FUNCTION TryConvert_BYTE_TO_TOD : BOOL
VAR_INPUT
	in : BYTE;
	out : REFERENCE TO TOD;
END_VAR

out := BYTE_TO_TOD(in);
TryConvert_BYTE_TO_TOD := TRUE;

END_FUNCTION

(* stored: Version 1.1.0.1, ProductVersion 3.1.4024.12
   POU TryConvert_BYTE_TO_TOD: Id {392e3d4e-3f2c-48fe-bc46-4599fb8bc015}, SpecialFunc None *)
